(* Schneider Machine Expert - Basic project 08_edges, file version 3.0.0.0 *)
(* ProjectInformations: Name=New project *)

HARDWARE
  Cpu 0: TM221C40R
  EthernetConfiguration: NetworkName=M221, IpAllocationMode=FixedAddress, IpAddress=0.0.0.0, SubnetMask=0.0.0.0
  SerialLineConfiguration: Baud=Baud19200, Parity=ParityEven, DataBits=DataBits8, StopBits=StopBits1, PhysicalMedium=PhysicalMediumRs485, TransmissionMode=TransmissionModeModbusRtu, SlaveId=1, Addressing=SlaveAddressing
  MastTask: UsePeriodScanMode=false, PeriodScan=100
  FastTask: Period=255
  CpuBehavior: StartingMode=StartAsPreviousState, AutoSaveRamOnEeprom=true, WatchdogPeriod=250

SYMBOLS  (address, symbol, comment, settings)

POU New POU
  (* SectionNumber=0 *)

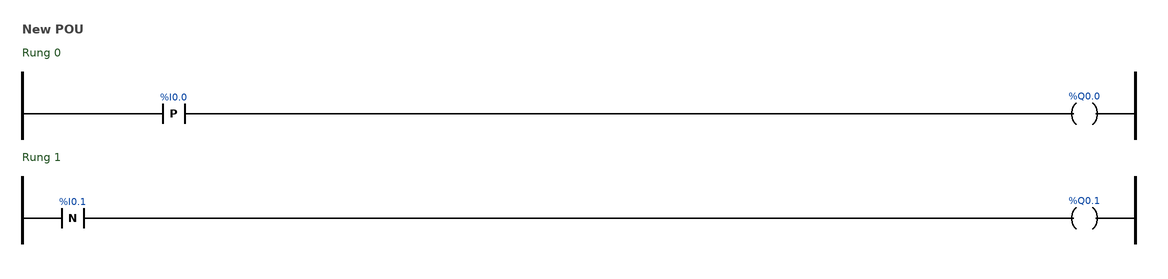

// Rung 0
  LDR %I0.0
  ST %Q0.0
  // as ST:
  //   %Q0.0 := RISING(%I0.0);

// Rung 1
  LDF %I0.1
  ST %Q0.1
  // as ST:
  //   %Q0.1 := FALLING(%I0.1);
